(* PLC project MC500_EtherCAT_axis_motion, LeadShine company LeadSys Studio V3.1.0.0 LeadSysStudio V3.5 SP15 Patch 4 *)
(* stored: creationDateTime 2026-07-01T11:09:49.0050075, modificationDateTime 2026-07-01T10:49:55.3800865 *)

PROGRAM MainSeq
  VAR
    fbGrid : GridCalc;  (* grid math, called in A_GridCalc *)
    griddle_dwell : TON;  (* A_Error, A_GriddleDwell, A_Idle *)
    grip_timer : TON;  (* A_Grip, A_Release *)
    loop_dwell : TON;  (* A_Wait *)
    GRIP_TIME : TIME := TIME#500ms;  (* time constants *)
    RELEASE_TIME : TIME := TIME#500ms;
    GRIDDLE_DWELL_T : TIME := TIME#5s0ms;
    LOOP_DWELL_T : TIME := TIME#3s0ms;
  END_VAR

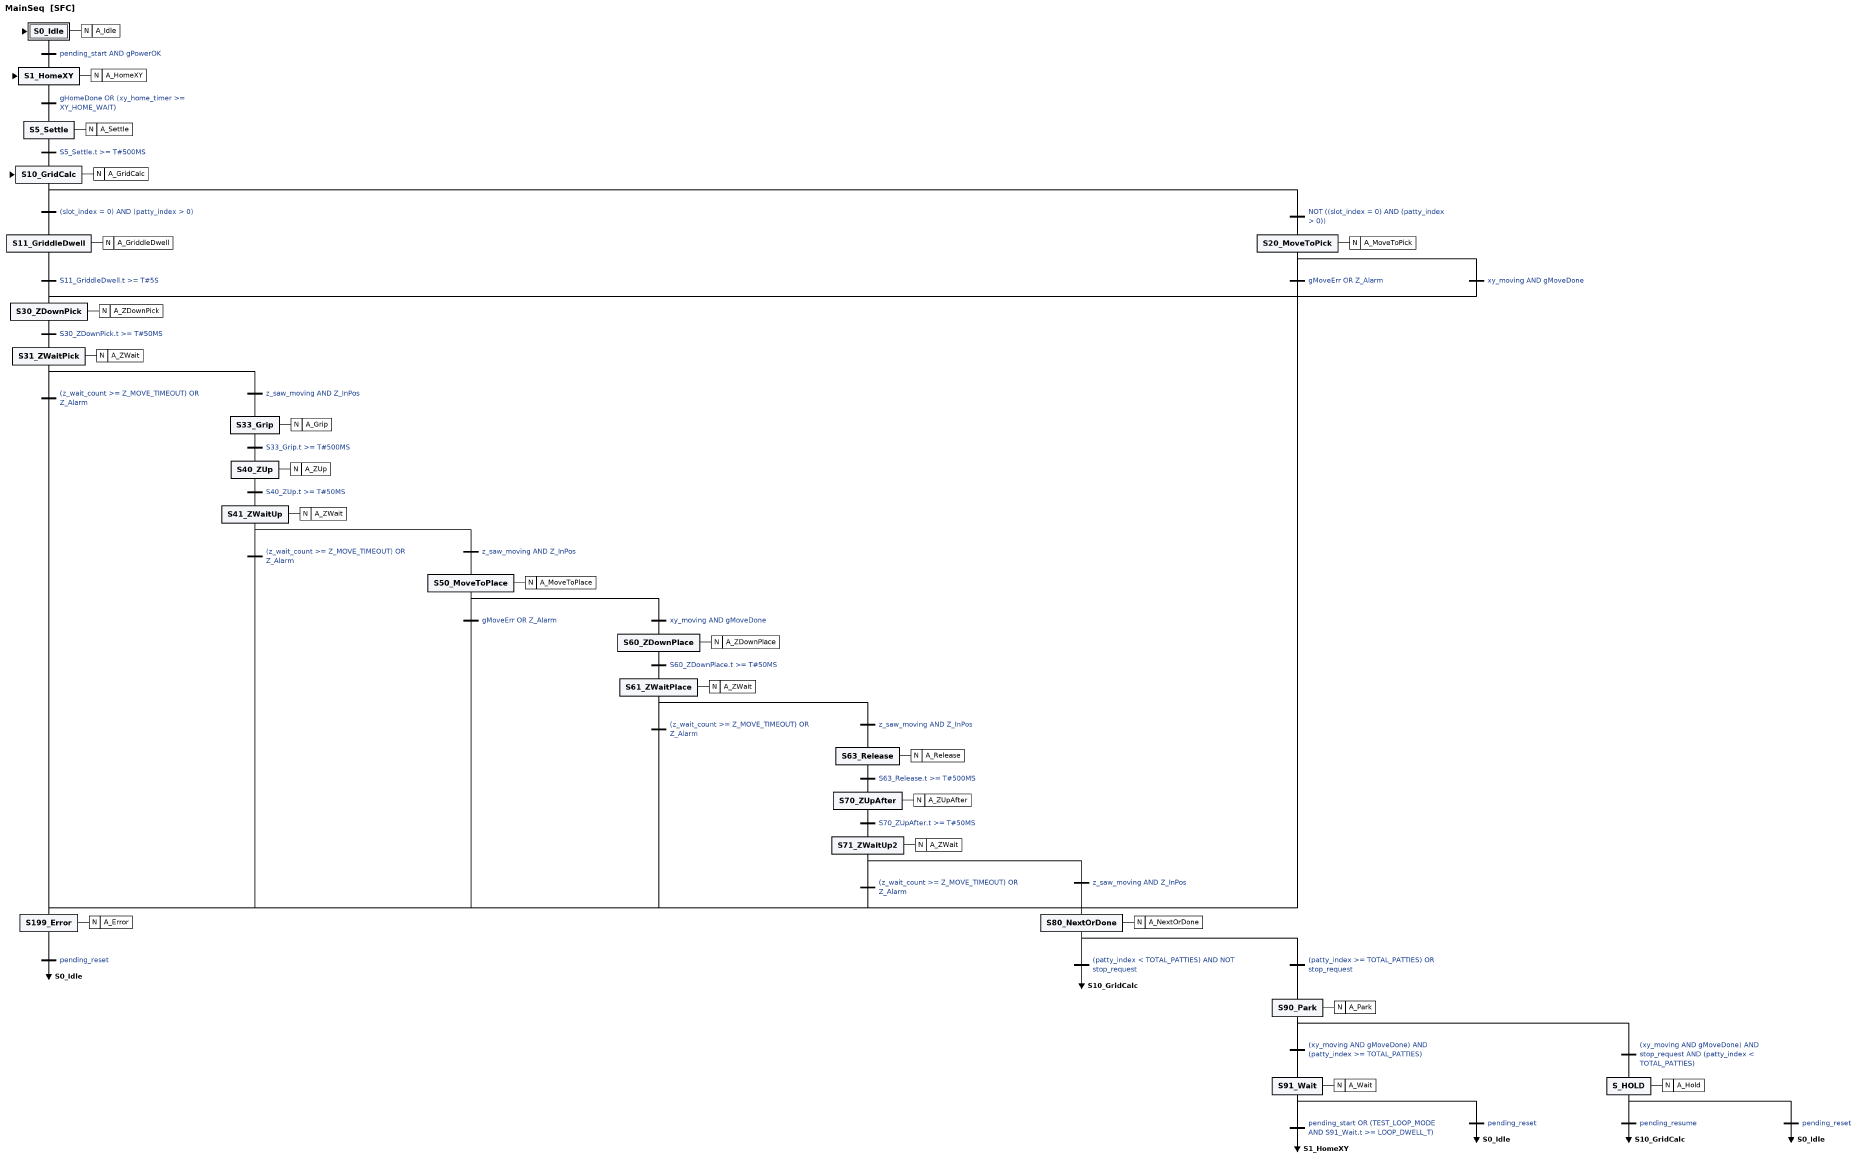
INITIAL_STEP S0_Idle:
  A_Idle(N);
END_STEP
TRANSITION FROM S0_Idle TO S1_HomeXY
  := pending_start AND gPowerOK;
END_TRANSITION
STEP S1_HomeXY:
  A_HomeXY(N);
END_STEP
TRANSITION FROM S1_HomeXY TO S5_Settle
  := gHomeDone OR (xy_home_timer >= XY_HOME_WAIT);
END_TRANSITION
STEP S5_Settle:
  A_Settle(N);
END_STEP
TRANSITION FROM S5_Settle TO S10_GridCalc
  := S5_Settle.t >= T#500MS;
END_TRANSITION
STEP S10_GridCalc:
  A_GridCalc(N);
END_STEP
TRANSITION FROM S10_GridCalc TO S11_GriddleDwell
  := (slot_index = 0) AND (patty_index > 0);
END_TRANSITION
TRANSITION FROM S10_GridCalc TO S20_MoveToPick
  := NOT ((slot_index = 0) AND (patty_index > 0));
END_TRANSITION
STEP S11_GriddleDwell:
  A_GriddleDwell(N);
END_STEP
TRANSITION FROM S11_GriddleDwell TO S30_ZDownPick
  := S11_GriddleDwell.t >= T#5S;
END_TRANSITION
STEP S20_MoveToPick:
  A_MoveToPick(N);
END_STEP
TRANSITION FROM S20_MoveToPick TO S199_Error
  := gMoveErr OR Z_Alarm;
END_TRANSITION
TRANSITION FROM S20_MoveToPick TO S30_ZDownPick
  := xy_moving AND gMoveDone;
END_TRANSITION
STEP S199_Error:
  A_Error(N);
END_STEP
TRANSITION FROM S199_Error TO S0_Idle
  := pending_reset;
END_TRANSITION
STEP S30_ZDownPick:
  A_ZDownPick(N);
END_STEP
TRANSITION FROM S30_ZDownPick TO S31_ZWaitPick
  := S30_ZDownPick.t >= T#50MS;
END_TRANSITION
STEP S31_ZWaitPick:
  A_ZWait(N);
END_STEP
TRANSITION FROM S31_ZWaitPick TO S199_Error
  := (z_wait_count >= Z_MOVE_TIMEOUT) OR Z_Alarm;
END_TRANSITION
TRANSITION FROM S31_ZWaitPick TO S33_Grip
  := z_saw_moving AND Z_InPos;
END_TRANSITION
STEP S33_Grip:
  A_Grip(N);
END_STEP
TRANSITION FROM S33_Grip TO S40_ZUp
  := S33_Grip.t >= T#500MS;
END_TRANSITION
STEP S40_ZUp:
  A_ZUp(N);
END_STEP
TRANSITION FROM S40_ZUp TO S41_ZWaitUp
  := S40_ZUp.t >= T#50MS;
END_TRANSITION
STEP S41_ZWaitUp:
  A_ZWait(N);
END_STEP
TRANSITION FROM S41_ZWaitUp TO S199_Error
  := (z_wait_count >= Z_MOVE_TIMEOUT) OR Z_Alarm;
END_TRANSITION
TRANSITION FROM S41_ZWaitUp TO S50_MoveToPlace
  := z_saw_moving AND Z_InPos;
END_TRANSITION
STEP S50_MoveToPlace:
  A_MoveToPlace(N);
END_STEP
TRANSITION FROM S50_MoveToPlace TO S199_Error
  := gMoveErr OR Z_Alarm;
END_TRANSITION
TRANSITION FROM S50_MoveToPlace TO S60_ZDownPlace
  := xy_moving AND gMoveDone;
END_TRANSITION
STEP S60_ZDownPlace:
  A_ZDownPlace(N);
END_STEP
TRANSITION FROM S60_ZDownPlace TO S61_ZWaitPlace
  := S60_ZDownPlace.t >= T#50MS;
END_TRANSITION
STEP S61_ZWaitPlace:
  A_ZWait(N);
END_STEP
TRANSITION FROM S61_ZWaitPlace TO S199_Error
  := (z_wait_count >= Z_MOVE_TIMEOUT) OR Z_Alarm;
END_TRANSITION
TRANSITION FROM S61_ZWaitPlace TO S63_Release
  := z_saw_moving AND Z_InPos;
END_TRANSITION
STEP S63_Release:
  A_Release(N);
END_STEP
TRANSITION FROM S63_Release TO S70_ZUpAfter
  := S63_Release.t >= T#500MS;
END_TRANSITION
STEP S70_ZUpAfter:
  A_ZUpAfter(N);
END_STEP
TRANSITION FROM S70_ZUpAfter TO S71_ZWaitUp2
  := S70_ZUpAfter.t >= T#50MS;
END_TRANSITION
STEP S71_ZWaitUp2:
  A_ZWait(N);
END_STEP
TRANSITION FROM S71_ZWaitUp2 TO S199_Error
  := (z_wait_count >= Z_MOVE_TIMEOUT) OR Z_Alarm;
END_TRANSITION
TRANSITION FROM S71_ZWaitUp2 TO S80_NextOrDone
  := z_saw_moving AND Z_InPos;
END_TRANSITION
STEP S80_NextOrDone:
  A_NextOrDone(N);
END_STEP
TRANSITION FROM S80_NextOrDone TO S10_GridCalc
  := (patty_index < TOTAL_PATTIES) AND NOT stop_request;
END_TRANSITION
TRANSITION FROM S80_NextOrDone TO S90_Park
  := (patty_index >= TOTAL_PATTIES) OR stop_request;
END_TRANSITION
STEP S90_Park:
  A_Park(N);
END_STEP
TRANSITION FROM S90_Park TO S91_Wait
  := (xy_moving AND gMoveDone) AND (patty_index >= TOTAL_PATTIES);
END_TRANSITION
TRANSITION FROM S90_Park TO S_HOLD
  := (xy_moving AND gMoveDone) AND stop_request AND (patty_index < TOTAL_PATTIES);
END_TRANSITION
STEP S_HOLD:
  A_Hold(N);
END_STEP
TRANSITION FROM S_HOLD TO S10_GridCalc
  := pending_resume;
END_TRANSITION
TRANSITION FROM S_HOLD TO S0_Idle
  := pending_reset;
END_TRANSITION
STEP S91_Wait:
  A_Wait(N);
END_STEP
TRANSITION FROM S91_Wait TO S1_HomeXY
  := pending_start OR (TEST_LOOP_MODE AND S91_Wait.t >= LOOP_DWELL_T);
END_TRANSITION
TRANSITION FROM S91_Wait TO S0_Idle
  := pending_reset;
END_TRANSITION

ACTION A_Idle:
                        state := 0;
cycle_complete := FALSE;  cycle_active := FALSE;  paused := FALSE;
end_effector := FALSE;
z_wait_count := 0;        xy_home_timer := 0;
griddle_index := 0;       slot_index := 0;
griddle_dwell(IN := FALSE);
gMoveExec := FALSE;  gHomeExec := FALSE;  gStopExec := FALSE;
xy_moving := FALSE;  np_done := FALSE;          // <-- add np_done here
Z_DO_Down := FALSE;  Z_Trig := FALSE;
stop_request := FALSE;  holding := FALSE;  pending_reset := FALSE;
                      
END_ACTION

ACTION A_HomeXY:
                        state := 1;
IF NOT cycle_active THEN
    pending_start := FALSE;        // ← drop the pending_restart line
    patty_index := 0;
	np_done := FALSE;  
  	cycle_active := TRUE;
END_IF
gHomeExec := TRUE;
xy_home_timer := xy_home_timer + 1;
IF gHomeDone OR (xy_home_timer >= XY_HOME_WAIT) THEN
    gHomeExec := FALSE;  xy_home_timer := 0;  z_wait_count := 0;
END_IF
                      
END_ACTION

ACTION A_GridCalc:
                        state := 10;
IF holding THEN
    holding := FALSE;
    stop_request := FALSE;
    pending_resume := FALSE;
    cycle_active := TRUE;
END_IF
fbGrid(idx := patty_index);
                      
END_ACTION

ACTION A_GriddleDwell:
                        state := 11;
griddle_dwell(IN := TRUE, PT := GRIDDLE_DWELL_T);
TargetXY[0] := pick_x;  TargetXY[1] := pick_y;     // travel to pick during rotation
gMoveExec := TRUE;
IF gMoveBusy OR NOT gMoveDone THEN xy_moving := TRUE; END_IF
IF griddle_dwell.Q THEN griddle_dwell(IN := FALSE); END_IF
                      
END_ACTION

ACTION A_MoveToPick:
                        state := 20;
TargetXY[0] := pick_x;  TargetXY[1] := pick_y;
gMoveExec := TRUE;
IF gMoveBusy OR NOT gMoveDone THEN xy_moving := TRUE; END_IF
                      
END_ACTION

ACTION A_Grip:
                        state := 33;
end_effector := TRUE;


                      
END_ACTION

ACTION A_MoveToPlace:
                        state := 50;
TargetXY[0] := place_x;  TargetXY[1] := place_y;
gMoveExec := TRUE;
IF gMoveBusy OR NOT gMoveDone THEN xy_moving := TRUE; END_IF
                      
END_ACTION

ACTION A_Release:
                        state := 63;
end_effector := FALSE;

                      
END_ACTION

ACTION A_NextOrDone:
                        state := 80;
IF NOT np_done THEN
    patty_index := patty_index + 1;
    np_done := TRUE;
END_IF
                      
END_ACTION

ACTION A_Park:
                        state := 90;
TargetXY[0] := 50.0;  TargetXY[1] := 50.0;
gMoveExec := TRUE;
IF gMoveBusy OR NOT gMoveDone THEN xy_moving := TRUE; END_IF
IF (xy_moving AND gMoveDone) OR gMoveErr THEN
    cycle_active := FALSE;
    IF patty_index >= TOTAL_PATTIES THEN
        cycle_complete := TRUE;
        cycle_count := cycle_count + 1;
    END_IF
END_IF
                      
END_ACTION

ACTION A_Wait:
                        state := 91;
gMoveExec := FALSE;  xy_moving := FALSE;      // release the park move
np_done := FALSE;                             // arm patty counter for next run
                      
END_ACTION

ACTION A_Settle:
                        state := 5;
  gHomeExec := FALSE;
  gMoveExec := FALSE;
                      
END_ACTION

ACTION A_Error:
                        state := 199;
gMoveExec := FALSE;
gHomeExec := FALSE;
gStopExec := FALSE;
end_effector := FALSE;
griddle_dwell(IN := FALSE);
 Z_DO_Down := FALSE;
                      
END_ACTION

ACTION A_Hold:
                        state := 95;
holding := TRUE;
cycle_active := FALSE;
gMoveExec := FALSE;  xy_moving := FALSE;
                      
END_ACTION

ACTION A_ZDownPick:
                        state := 30;
gMoveExec := FALSE;  xy_moving := FALSE;     // release the pick move
Z_DO_Down := TRUE;   Z_Trig := FALSE;        // select down path, CTRG low
z_saw_moving := FALSE;  z_wait_count := 0;
                      
END_ACTION

ACTION A_ZUp:
                        state:=40; Z_DO_Down := FALSE; Z_Trig := FALSE; z_saw_moving:=FALSE; z_wait_count:=0;
                      
END_ACTION

ACTION A_ZDownPlace:
                        state := 60;
gMoveExec := FALSE;  xy_moving := FALSE;     // release the place move
Z_DO_Down := TRUE;   Z_Trig := FALSE;
z_saw_moving := FALSE;  z_wait_count := 0;
                      
END_ACTION

ACTION A_ZUpAfter:
                        state := 70;
gMoveExec := FALSE;  xy_moving := FALSE;     // (if you added these — keep)
Z_DO_Down := FALSE;  Z_Trig := FALSE;
z_saw_moving := FALSE;  z_wait_count := 0;
np_done := FALSE;                            // arm the one-shot for S80
                      
END_ACTION

ACTION A_ZWait:
                        Z_Trig := TRUE;                 // rising edge (address was set last step) -> executes selected path
z_wait_count := z_wait_count + 1;
IF NOT Z_InPos THEN
    z_saw_moving := TRUE;
END_IF
                      
END_ACTION
END_PROGRAM

PROGRAM PLC_PRG

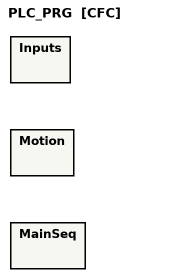
(* CFC diagram, written out as Structured Text *)
Inputs();
Motion();
MainSeq();
END_PROGRAM

PROGRAM Inputs
  VAR
    btn_a AT %IX0.0 : BOOL;
    btn_b AT %IX0.1 : BOOL;
    btn_reset AT %IX0.2 : BOOL;  (* physical Reset (wire later) *)
  END_VAR
  VAR
    rt_a : R_TRIG;
    rt_b : R_TRIG;
    edgeA : BOOL;
    edgeB : BOOL;
    rt_reset : R_TRIG;
    edgeReset : BOOL;
  END_VAR

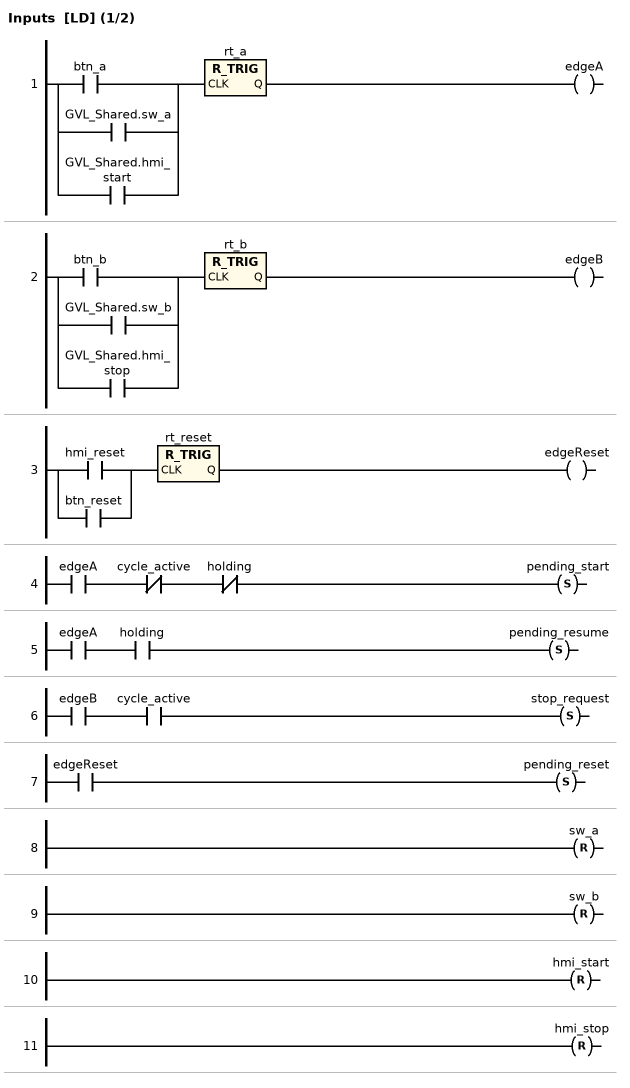
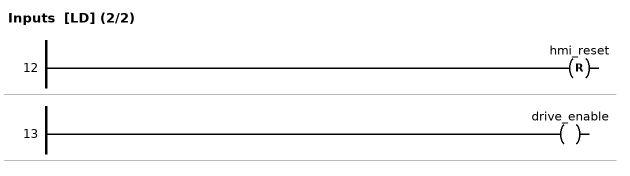
(* LD diagram, written out as Structured Text *)
(* --- network: ...... --- *)
rt_a(CLK := btn_a OR GVL_Shared.sw_a OR GVL_Shared.hmi_start);
edgeA := rt_a.Q;
(* NetworkDefaultComment *)
(* --- network: ...... --- *)
rt_b(CLK := btn_b OR GVL_Shared.sw_b OR GVL_Shared.hmi_stop);
edgeB := rt_b.Q;
(* NetworkDefaultComment *)
(* --- network: ...... --- *)
rt_reset(CLK := hmi_reset OR btn_reset);
edgeReset := rt_reset.Q;
(* NetworkDefaultComment *)
(* --- network: ...... --- *)
IF edgeA AND NOT cycle_active AND NOT holding THEN pending_start := TRUE; END_IF;
(* NetworkDefaultComment *)
(* --- network: ...... --- *)
IF edgeA AND holding THEN pending_resume := TRUE; END_IF;
(* NetworkDefaultComment *)
(* --- network: ...... --- *)
IF edgeB AND cycle_active THEN stop_request := TRUE; END_IF;
(* NetworkDefaultComment *)
(* --- network: ...... --- *)
IF edgeReset THEN pending_reset := TRUE; END_IF;
(* NetworkDefaultComment *)
(* --- network: ...... --- *)
IF TRUE THEN sw_a := FALSE; END_IF;
IF TRUE THEN sw_b := FALSE; END_IF;
IF TRUE THEN hmi_start := FALSE; END_IF;
IF TRUE THEN hmi_stop := FALSE; END_IF;
IF TRUE THEN hmi_reset := FALSE; END_IF;
(* NetworkDefaultComment *)
(* --- network: ...... --- *)
drive_enable := TRUE;
END_PROGRAM

PROGRAM Motion
  VAR
    MC_Power_1 : MC_Power;
    MC_Power_2 : MC_Power;
    MC_Home_1 : MC_Home;
    MC_Home_2 : MC_Home;
    MC_Stop_1 : MC_Stop;
    MC_Stop_2 : MC_Stop;
    MC_Reset_1 : MC_Reset;
    LS_MOVEXY : LS_2AxisLine;
    MC_Reset_2 : MC_Reset;
  END_VAR
  VAR  (* added by the conversion: wires and edge detectors of the diagram *)
    _AND11_OUT : BOOL;
  END_VAR

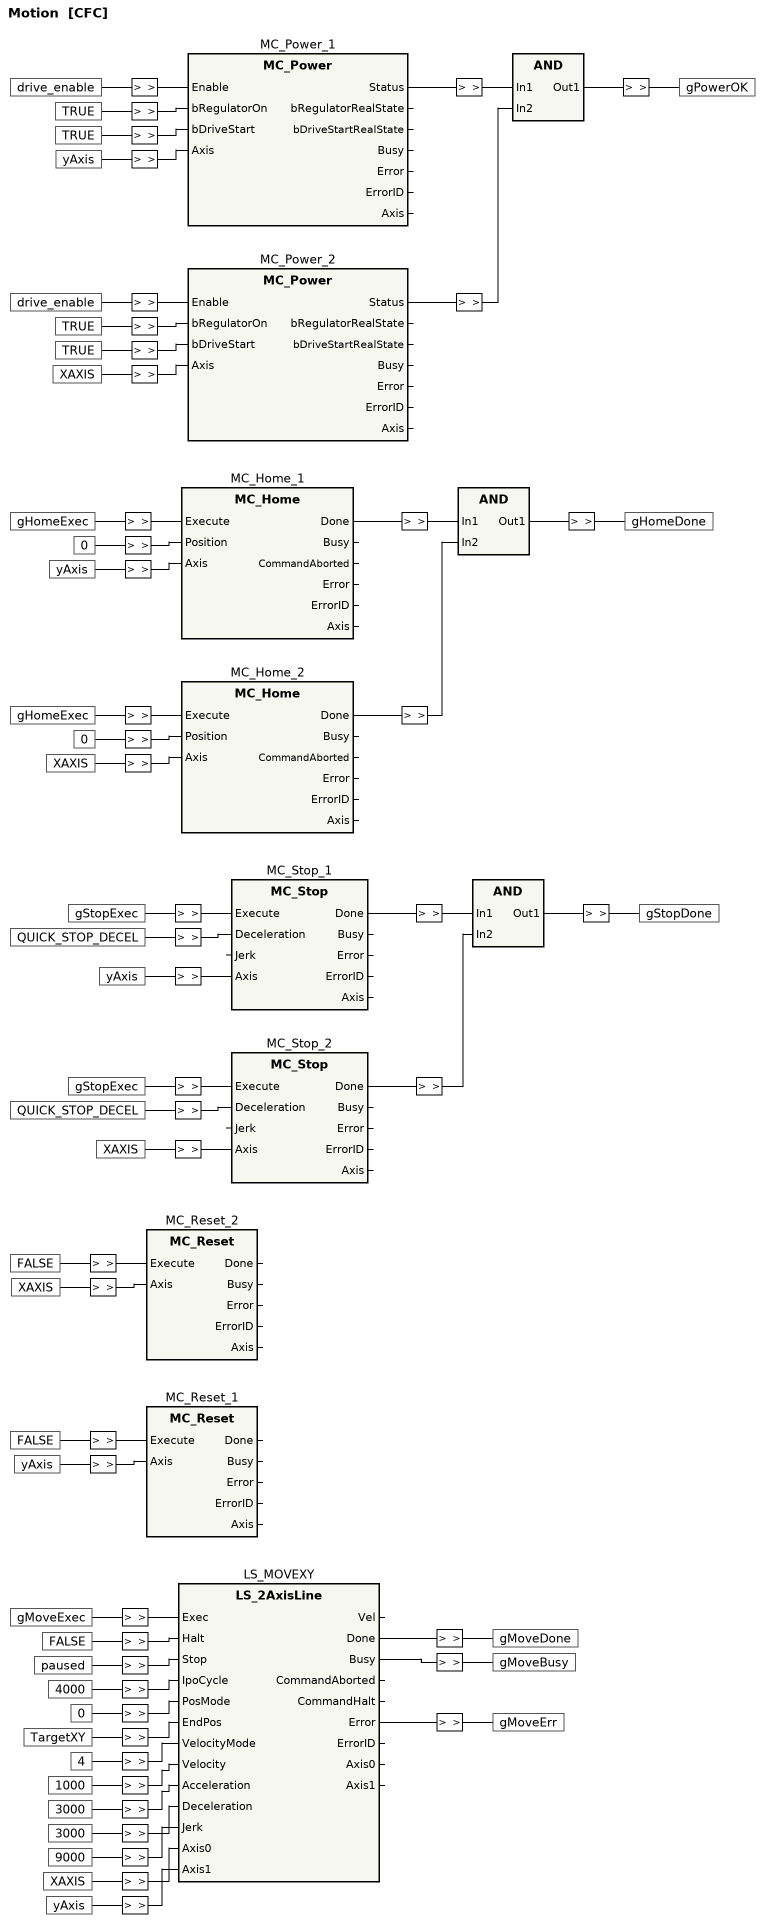
(* CFC diagram, written out as Structured Text *)
MC_Power_2(Enable := drive_enable, bRegulatorOn := TRUE, bDriveStart := TRUE, Axis := XAXIS);
gHomeDone := _AND11_OUT;
MC_Home_2(Execute := gHomeExec, Position := 0, Axis := XAXIS);
MC_Stop_2(Execute := gStopExec, Deceleration := QUICK_STOP_DECEL, Axis := XAXIS);
MC_Power_1(Enable := drive_enable, bRegulatorOn := TRUE, bDriveStart := TRUE, Axis := yAxis);
gPowerOK := MC_Power_1.Status AND MC_Power_2.Status;
MC_Home_1(Execute := gHomeExec, Position := 0, Axis := yAxis);
_AND11_OUT := MC_Home_1.Done AND MC_Home_2.Done;
MC_Reset_2(Execute := FALSE, Axis := XAXIS);
MC_Stop_1(Execute := gStopExec, Deceleration := QUICK_STOP_DECEL, Axis := yAxis);
gStopDone := MC_Stop_1.Done AND MC_Stop_2.Done;
MC_Reset_1(Execute := FALSE, Axis := yAxis);
gMoveDone := LS_MOVEXY.Done;
LS_MOVEXY(Exec := gMoveExec, Halt := FALSE, Stop := paused, IpoCycle := 4000, PosMode := 0, EndPos := TargetXY, VelocityMode := 4, Velocity := 1000, Acceleration := 3000, Deceleration := 3000, Jerk := 9000, Axis0 := XAXIS, Axis1 := yAxis);
gMoveBusy := LS_MOVEXY.Busy;
gMoveErr := LS_MOVEXY.Error;
END_PROGRAM

(* ---- DECLARATION pane ---- *)
FUNCTION_BLOCK GridCalc
  VAR_INPUT
    idx : INT;  (* = patty_index *)
  END_VAR

                    
current_row := idx / TRAY_COLS;
current_col := idx MOD TRAY_COLS;
pick_x := PICK_BASE_X + INT_TO_LREAL(current_col) * PICK_SPACING_X;
pick_y := PICK_BASE_Y + INT_TO_LREAL(current_row) * PICK_SPACING_Y;
 
griddle_index := idx / PATTIES_PER_GRIDDLE;
slot_index    := idx MOD PATTIES_PER_GRIDDLE;
place_x := PLACE_BASE_X + PLACE_OFFSET_X[slot_index];
place_y := PLACE_BASE_Y + PLACE_OFFSET_Y[slot_index];
 
                  
END_FUNCTION_BLOCK

CONFIGURATION Device
  RESOURCE Application ON PLC
    VAR_GLOBAL  (* GVL_Shared - ===================================================================== GVL "GVL_Shared" — globals shared across the LD / CFC / SFC / ST POUs (Splitting one POU into four means the formerly-local VARs become globals grouped by owner. Comment // [owner->reader] shows the data direction.) ===================================================================== *)
      pending_start : BOOL := FALSE;  (* ---- AXIS REFERENCES (declared in your hardware config) ---- XAXIS, yAxis : AXIS_REF; // already exist in the project ============ COMMAND FLAGS : LD (Inputs) -> SFC ============ *)
      pending_resume : BOOL := FALSE;
      hmi_start : BOOL := FALSE;  (* HMI write *)
      sw_a : BOOL := FALSE;  (* HMI/soft button A *)
      sw_b : BOOL := FALSE;  (* HMI/soft button B *)
      gMoveExec : BOOL := FALSE;  (* drive LS_MoveXY.Exec *)
      gHomeExec : BOOL := FALSE;  (* drive MC_Home_1/2.Execute *)
      gStopExec : BOOL := FALSE;  (* drive MC_Stop_1/2.Execute *)
      TargetXY : ARRAY[0..1] OF LREAL := [0.0, 0.0];
      drive_enable : BOOL := TRUE;  (* MC_Power_*.Enable (set by Inputs/Pause) *)
      gPowerOK : BOOL := FALSE;  (* MC_Power_1.Status AND MC_Power_2.Status *)
      gMoveDone : BOOL := FALSE;  (* LS_MoveXY.Done *)
      gMoveErr : BOOL := FALSE;  (* LS_MoveXY.Error *)
      gMoveBusy : BOOL := FALSE;  (* LS_MoveXY.Busy *)
      gHomeDone : BOOL := FALSE;  (* MC_Home_1.Done AND MC_Home_2.Done *)
      gStopDone : BOOL := FALSE;  (* MC_Stop_1.Done AND MC_Stop_2.Done *)
      end_effector AT %QX1.4 : BOOL := FALSE;  (* LD coil *)
      QUICK_STOP_DECEL : LREAL := 3000.0;
      PICK_BASE_X : LREAL := 145.0;  (* ============ Z AXIS — MODBUS I/O (CS2RS-D1008) ============= ============ TRAY / GRID CONFIG (read by GridCalc) ======== *)
      PICK_BASE_Y : LREAL := 45.0;
      PICK_SPACING_X : LREAL := 80.0;
      PICK_SPACING_Y : LREAL := 80.0;
      PLACE_BASE_X : LREAL := 740.0;
      PLACE_BASE_Y : LREAL := 116.0;
      PLACE_OFFSET_X : ARRAY[0..5] OF LREAL := [0.0, 70.0, -70.0, 70.0, -70.0, 0.0];
      PLACE_OFFSET_Y : ARRAY[0..5] OF LREAL := [0.0, 66.0, 66.0, 143.0, 143.0, 210.0];
      TRAY_COLS : INT := 6;
      TRAY_ROWS : INT := 4;
      TOTAL_PATTIES : INT := 24;
      PATTIES_PER_GRIDDLE : INT := 6;
      GRIDDLE_COUNT : INT := 4;
      patty_index : INT := 0;  (* ============ GRID RESULTS (GridCalc -> SFC) =============== *)
      current_col : INT := 0;
      current_row : INT := 0;
      griddle_index : INT := 0;
      slot_index : INT := 0;
      pick_x : LREAL := 0.0;
      pick_y : LREAL := 0.0;
      place_x : LREAL := 0.0;
      place_y : LREAL := 0.0;
      TEST_LOOP_MODE : BOOL := TRUE;  (* ============ MODE / BOOKKEEPING =========================== *)
      cycle_count : UDINT := 0;
      cycle_complete : BOOL := FALSE;
      cycle_active : BOOL := FALSE;
      paused : BOOL := FALSE;
      XY_HOME_WAIT : INT := 7500;  (* ============ TIMING CONSTANTS ============================= *)
      xy_home_timer : INT := 0;
      stop_request : BOOL := FALSE;  (* CYCLE-stop request (operator Stop button) *)
      holding : BOOL := FALSE;  (* TRUE while parked & held *)
      pending_reset : BOOL := FALSE;
      hmi_stop : BOOL := FALSE;
      hmi_reset : BOOL := FALSE;
      Z_DO_Down AT %QX1.5 : BOOL := FALSE;  (* pulse -> down path *)
      Z_InPos AT %IX1.0 : BOOL;  (* SO1 INP = positioning complete *)
      z_saw_moving : BOOL := FALSE;
      Z_Alarm AT %IX1.1 : BOOL;  (* SO3 ALM (check polarity) *)
      z_wait_count : INT := 0;
      Z_MOVE_TIMEOUT : INT := 2500;
      state : INT := 0;
      Z_Disable AT %QX1.3 : BOOL := FALSE;  (* TRUE = disable Z drive; FALSE (default) = enabled *)
      Z_Trig AT %QX1.6 : BOOL := FALSE;
      xy_moving : BOOL := FALSE;
      np_done : BOOL := FALSE;
    END_VAR
    TASK MainTask(INTERVAL := T#4ms, PRIORITY := 1);
    PROGRAM EtherCAT_Master_Leadshine_A.EtherCAT_Task WITH MainTask : EtherCAT_Master_Leadshine_A.EtherCAT_Task;
    PROGRAM PLC_PRG WITH MainTask : PLC_PRG;
  END_RESOURCE
END_CONFIGURATION

CONFIGURATION High_Speed_IO_Module
END_CONFIGURATION

CONFIGURATION LocalBus_Master_Module
END_CONFIGURATION

CONFIGURATION EtherCAT_Master_Leadshine_A
END_CONFIGURATION

CONFIGURATION CS3E_D1008_1
END_CONFIGURATION

CONFIGURATION XAXIS
END_CONFIGURATION

CONFIGURATION CS3E_D1008
END_CONFIGURATION

CONFIGURATION yAxis
END_CONFIGURATION

CONFIGURATION ModbusTCP_Slave_Device
END_CONFIGURATION

CONFIGURATION SoftMotion General Axis Pool
END_CONFIGURATION
